SYSTEM SystemTests
  (* Version 1.0, 2018-08-29, Alois Zoitl, Johannes Kepler University, initial API and implementation and/or initial documentation *)
  APPLICATION Timing (* Small test application for measuring the execution time of a few fbs for evaluating runtime performance *)
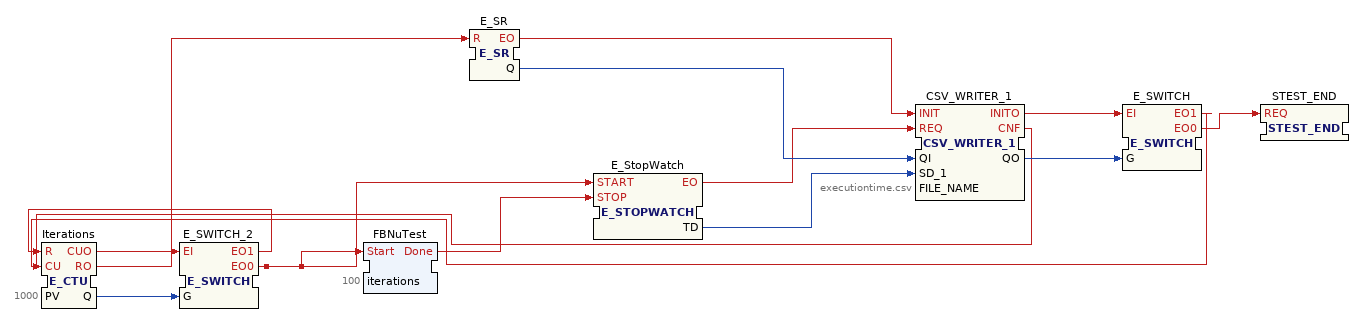
    FBS
      CSV_WRITER_1 : CSV_WRITER_1(FILE_NAME := executiontime.csv);
      E_SR : E_SR;
      E_SWITCH_2 : E_SWITCH;
      Iterations : E_CTU(PV := 1000);
      STEST_END : STEST_END;
      E_SWITCH : E_SWITCH;
      E_StopWatch : E_STOPWATCH;
    END_FBS
    SUBAPPLICATION FBNuTest(iterations := 100)
      EVENT_INPUT
        Start;
      END_EVENT
      EVENT_OUTPUT
        Done;
      END_EVENT
      VAR_INPUT
        iterations : UINT := 100;
      END_VAR
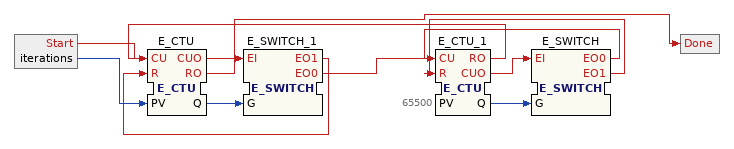
      FBS
        E_CTU : E_CTU;
        E_SWITCH_1 : E_SWITCH;
        E_SWITCH : E_SWITCH;
        E_CTU_1 : E_CTU(PV := 65500);
      END_FBS
      EVENT_CONNECTIONS
        E_CTU_1.RO TO E_CTU.CU;
        E_SWITCH_1.EO1 TO E_CTU.R;
        E_CTU.CUO TO E_SWITCH_1.EI;
        E_SWITCH_1.EO0 TO E_CTU_1.CU;
        E_CTU_1.CUO TO E_SWITCH.EI;
        E_SWITCH.EO0 TO E_CTU_1.CU;
        E_SWITCH.EO1 TO E_CTU_1.R;
        Start TO E_CTU.CU;
        E_CTU.RO TO Done;
      END_CONNECTIONS
      DATA_CONNECTIONS
        E_CTU.Q TO E_SWITCH_1.G;
        E_CTU_1.Q TO E_SWITCH.G;
        iterations TO E_CTU.PV;
      END_CONNECTIONS
    END_SUBAPPLICATION
    EVENT_CONNECTIONS
      E_SR.EO TO CSV_WRITER_1.INIT;
      Iterations.CUO TO E_SWITCH_2.EI;
      E_SWITCH_2.EO1 TO Iterations.R;
      Iterations.RO TO E_SR.R;
      E_SWITCH_2.EO0 TO FBNuTest.Start;
      E_SWITCH.EO1 TO Iterations.CU;
      E_SWITCH.EO0 TO STEST_END.REQ;
      CSV_WRITER_1.INITO TO E_SWITCH.EI;
      E_SWITCH_2.EO0 TO E_StopWatch.START;
      FBNuTest.Done TO E_StopWatch.STOP;
      E_StopWatch.EO TO CSV_WRITER_1.REQ;
      CSV_WRITER_1.CNF TO Iterations.CU;
    END_CONNECTIONS
    DATA_CONNECTIONS
      E_SR.Q TO CSV_WRITER_1.QI;
      Iterations.Q TO E_SWITCH_2.G;
      CSV_WRITER_1.QO TO E_SWITCH.G;
      E_StopWatch.TD TO CSV_WRITER_1.SD_1;
    END_CONNECTIONS
  END_APPLICATION
  APPLICATION Soft_Pass_Example
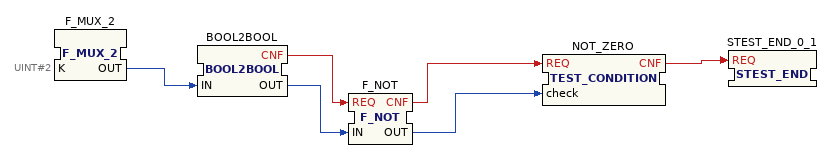
    FBS
      NOT_ZERO : TEST_CONDITION;
      STEST_END_0_1 : STEST_END;
      F_MUX_2 : F_MUX_2(K := UINT#2);
      F_NOT : F_NOT;
      BOOL2BOOL : BOOL2BOOL;
    END_FBS
    EVENT_CONNECTIONS
      F_NOT.CNF TO NOT_ZERO.REQ;
      NOT_ZERO.CNF TO STEST_END_0_1.REQ;
      BOOL2BOOL.CNF TO F_NOT.REQ;
    END_CONNECTIONS
    DATA_CONNECTIONS
      F_MUX_2.OUT TO BOOL2BOOL.IN;
      F_NOT.OUT TO NOT_ZERO.check;
      BOOL2BOOL.OUT TO F_NOT.IN;
    END_CONNECTIONS
  END_APPLICATION
  APPLICATION Fail_Example
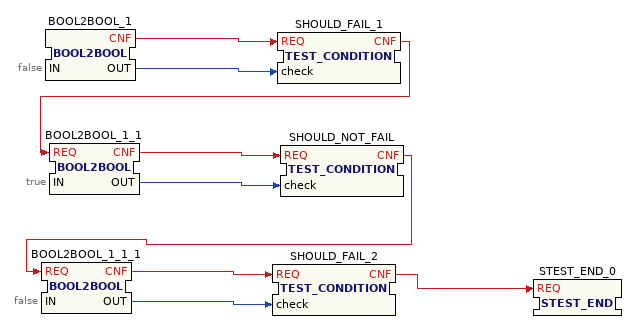
    FBS
      STEST_END_0 : STEST_END;
      BOOL2BOOL_1_1_1 : BOOL2BOOL(IN := false);
      SHOULD_FAIL_1 : TEST_CONDITION;
      BOOL2BOOL_1 : BOOL2BOOL(IN := false);
      SHOULD_NOT_FAIL : TEST_CONDITION;
      BOOL2BOOL_1_1 : BOOL2BOOL(IN := true);
      SHOULD_FAIL_2 : TEST_CONDITION;
    END_FBS
    EVENT_CONNECTIONS
      BOOL2BOOL_1.CNF TO SHOULD_FAIL_1.REQ;
      SHOULD_FAIL_2.CNF TO STEST_END_0.REQ;
      SHOULD_FAIL_1.CNF TO BOOL2BOOL_1_1.REQ;
      SHOULD_NOT_FAIL.CNF TO BOOL2BOOL_1_1_1.REQ;
      BOOL2BOOL_1_1_1.CNF TO SHOULD_FAIL_2.REQ;
      BOOL2BOOL_1_1.CNF TO SHOULD_NOT_FAIL.REQ;
    END_CONNECTIONS
    DATA_CONNECTIONS
      BOOL2BOOL_1_1.OUT TO SHOULD_NOT_FAIL.check;
      BOOL2BOOL_1.OUT TO SHOULD_FAIL_1.check;
      BOOL2BOOL_1_1_1.OUT TO SHOULD_FAIL_2.check;
    END_CONNECTIONS
  END_APPLICATION
  APPLICATION Hard_Pass_Example
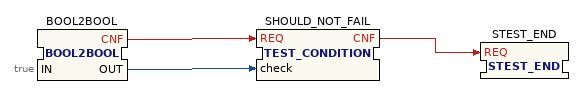
    FBS
      STEST_END : STEST_END;
      BOOL2BOOL : BOOL2BOOL(IN := true);
      SHOULD_NOT_FAIL : TEST_CONDITION;
    END_FBS
    EVENT_CONNECTIONS
      BOOL2BOOL.CNF TO SHOULD_NOT_FAIL.REQ;
      SHOULD_NOT_FAIL.CNF TO STEST_END.REQ;
    END_CONNECTIONS
    DATA_CONNECTIONS
      BOOL2BOOL.OUT TO SHOULD_NOT_FAIL.check;
    END_CONNECTIONS
  END_APPLICATION
  APPLICATION DeInitCommFB
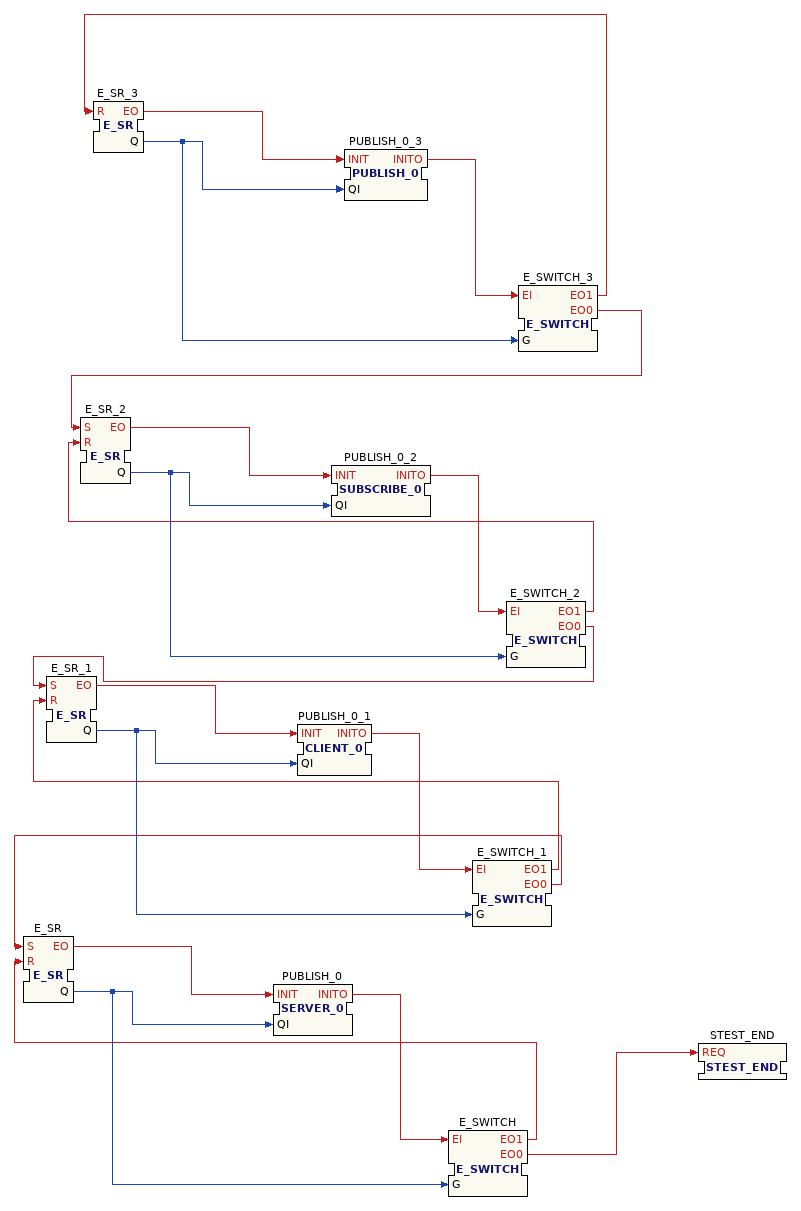
    FBS
      E_SR : E_SR;
      E_SWITCH : E_SWITCH;
      STEST_END : STEST_END;
      PUBLISH_0 : SERVER_0;
      E_SWITCH_1 : E_SWITCH;
      E_SR_1 : E_SR;
      E_SWITCH_2 : E_SWITCH;
      E_SR_2 : E_SR;
      E_SR_3 : E_SR;
      E_SWITCH_3 : E_SWITCH;
      PUBLISH_0_3 : PUBLISH_0;
      PUBLISH_0_2 : SUBSCRIBE_0;
      PUBLISH_0_1 : CLIENT_0;
    END_FBS
    EVENT_CONNECTIONS
      PUBLISH_0.INITO TO E_SWITCH.EI;
      E_SR_3.EO TO PUBLISH_0_3.INIT;
      PUBLISH_0_3.INITO TO E_SWITCH_3.EI;
      E_SR_2.EO TO PUBLISH_0_2.INIT;
      PUBLISH_0_2.INITO TO E_SWITCH_2.EI;
      E_SR_1.EO TO PUBLISH_0_1.INIT;
      PUBLISH_0_1.INITO TO E_SWITCH_1.EI;
      E_SWITCH_3.EO1 TO E_SR_3.R;
      E_SWITCH_3.EO0 TO E_SR_2.S;
      E_SWITCH_2.EO1 TO E_SR_2.R;
      E_SWITCH_2.EO0 TO E_SR_1.S;
      E_SWITCH_1.EO1 TO E_SR_1.R;
      E_SWITCH_1.EO0 TO E_SR.S;
      E_SWITCH.EO1 TO E_SR.R;
      E_SWITCH.EO0 TO STEST_END.REQ;
      E_SR.EO TO PUBLISH_0.INIT;
    END_CONNECTIONS
    DATA_CONNECTIONS
      E_SR.Q TO E_SWITCH.G;
      E_SR.Q TO PUBLISH_0.QI;
      E_SR_1.Q TO E_SWITCH_1.G;
      E_SR_2.Q TO E_SWITCH_2.G;
      E_SR_3.Q TO E_SWITCH_3.G;
      E_SR_3.Q TO PUBLISH_0_3.QI;
      E_SR_2.Q TO PUBLISH_0_2.QI;
      E_SR_1.Q TO PUBLISH_0_1.QI;
    END_CONNECTIONS
  END_APPLICATION
  APPLICATION simpleCommunicationTest
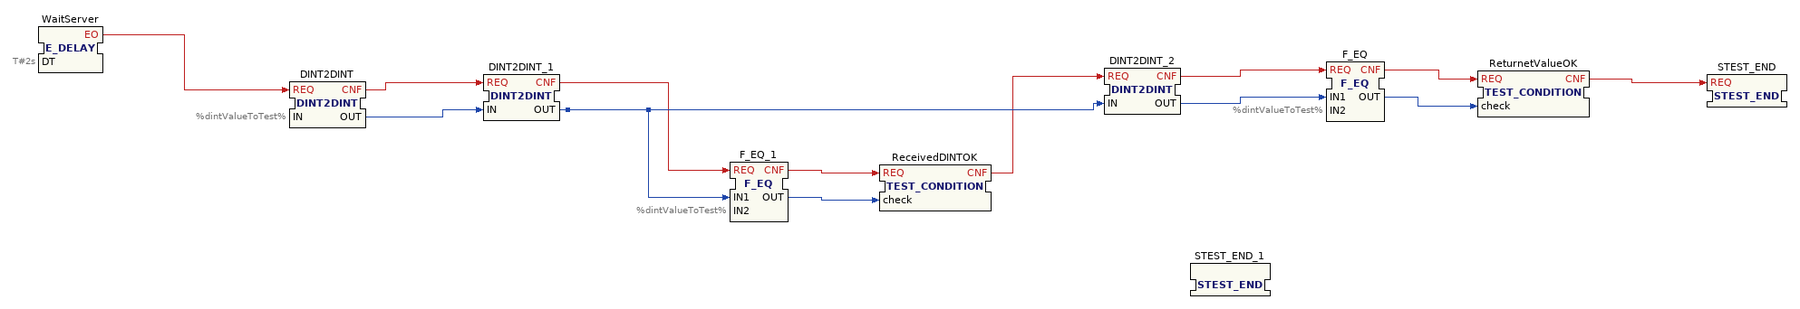
    FBS
      WaitServer : E_DELAY(DT := T#2s);
      ReturnetValueOK : TEST_CONDITION;
      F_EQ_1 : F_EQ(IN2 := %dintValueToTest%);
      F_EQ : F_EQ(IN2 := %dintValueToTest%);
      DINT2DINT_2 : DINT2DINT;
      DINT2DINT_1 : DINT2DINT;
      STEST_END : STEST_END;
      DINT2DINT : DINT2DINT(IN := %dintValueToTest%);
      ReceivedDINTOK : TEST_CONDITION;
      STEST_END_1 : STEST_END;
    END_FBS
    EVENT_CONNECTIONS
      DINT2DINT_1.CNF TO F_EQ_1.REQ;
      DINT2DINT.CNF TO DINT2DINT_1.REQ;
      ReceivedDINTOK.CNF TO DINT2DINT_2.REQ;
      F_EQ_1.CNF TO ReceivedDINTOK.REQ;
      F_EQ.CNF TO ReturnetValueOK.REQ;
      ReturnetValueOK.CNF TO STEST_END.REQ;
      DINT2DINT_2.CNF TO F_EQ.REQ;
      WaitServer.EO TO DINT2DINT.REQ;
    END_CONNECTIONS
    DATA_CONNECTIONS
      F_EQ_1.OUT TO ReceivedDINTOK.check;
      DINT2DINT_1.OUT TO DINT2DINT_2.IN;
      DINT2DINT.OUT TO DINT2DINT_1.IN;
      F_EQ.OUT TO ReturnetValueOK.check;
      DINT2DINT_1.OUT TO F_EQ_1.IN1;
      DINT2DINT_2.OUT TO F_EQ.IN1;
    END_CONNECTIONS
  END_APPLICATION
  APPLICATION CSVWriterTests
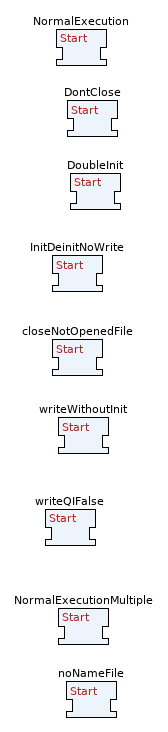
    SUBAPPLICATION NormalExecution
      EVENT_INPUT
        Start;
      END_EVENT
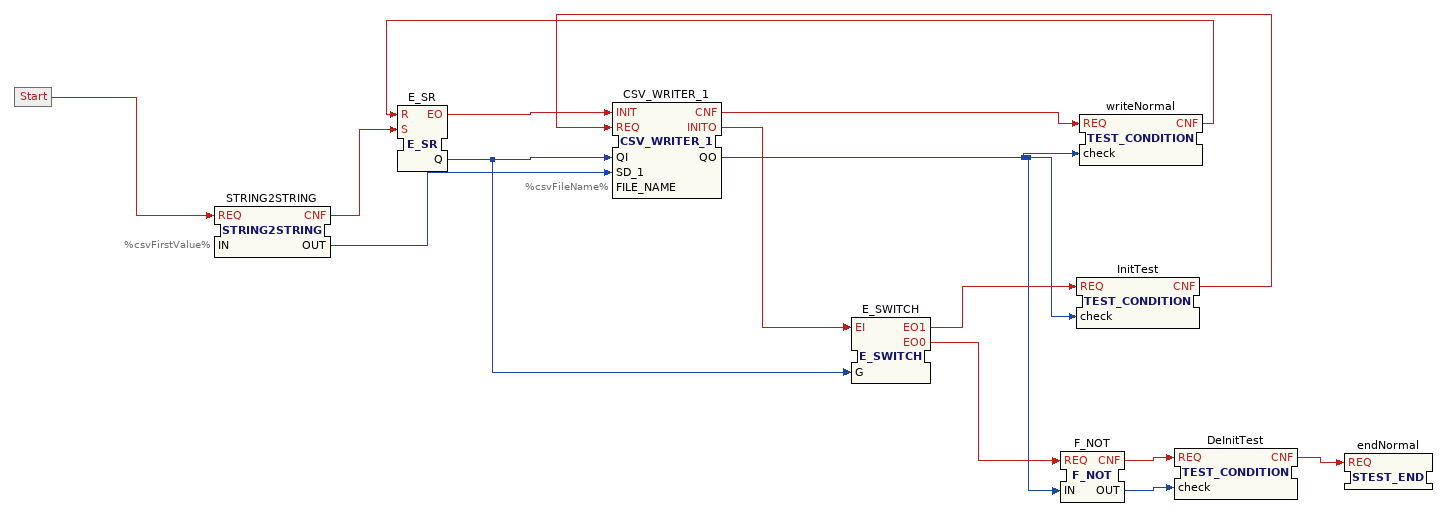
      FBS
        writeNormal : TEST_CONDITION;
        CSV_WRITER_1 : CSV_WRITER_1(FILE_NAME := %csvFileName%);
        InitTest : TEST_CONDITION;
        STRING2STRING : STRING2STRING(IN := %csvFirstValue%);
        DeInitTest : TEST_CONDITION;
        endNormal : STEST_END;
        F_NOT : F_NOT;
        E_SWITCH : E_SWITCH;
        E_SR : E_SR;
      END_FBS
      EVENT_CONNECTIONS
        CSV_WRITER_1.CNF TO writeNormal.REQ;
        writeNormal.CNF TO E_SR.R;
        E_SR.EO TO CSV_WRITER_1.INIT;
        InitTest.CNF TO CSV_WRITER_1.REQ;
        CSV_WRITER_1.INITO TO E_SWITCH.EI;
        E_SWITCH.EO1 TO InitTest.REQ;
        STRING2STRING.CNF TO E_SR.S;
        F_NOT.CNF TO DeInitTest.REQ;
        DeInitTest.CNF TO endNormal.REQ;
        E_SWITCH.EO0 TO F_NOT.REQ;
        Start TO STRING2STRING.REQ;
      END_CONNECTIONS
      DATA_CONNECTIONS
        CSV_WRITER_1.QO TO writeNormal.check;
        E_SR.Q TO CSV_WRITER_1.QI;
        STRING2STRING.OUT TO CSV_WRITER_1.SD_1;
        CSV_WRITER_1.QO TO InitTest.check;
        CSV_WRITER_1.QO TO F_NOT.IN;
        F_NOT.OUT TO DeInitTest.check;
        E_SR.Q TO E_SWITCH.G;
      END_CONNECTIONS
    END_SUBAPPLICATION
    SUBAPPLICATION DontClose
      EVENT_INPUT
        Start;
      END_EVENT
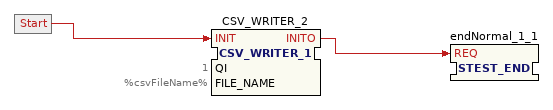
      FBS
        CSV_WRITER_2 : CSV_WRITER_1(QI := 1, FILE_NAME := %csvFileName%);
        endNormal_1_1 : STEST_END;
      END_FBS
      EVENT_CONNECTIONS
        CSV_WRITER_2.INITO TO endNormal_1_1.REQ;
        Start TO CSV_WRITER_2.INIT;
      END_CONNECTIONS
    END_SUBAPPLICATION
    SUBAPPLICATION DoubleInit
      EVENT_INPUT
        Start;
      END_EVENT
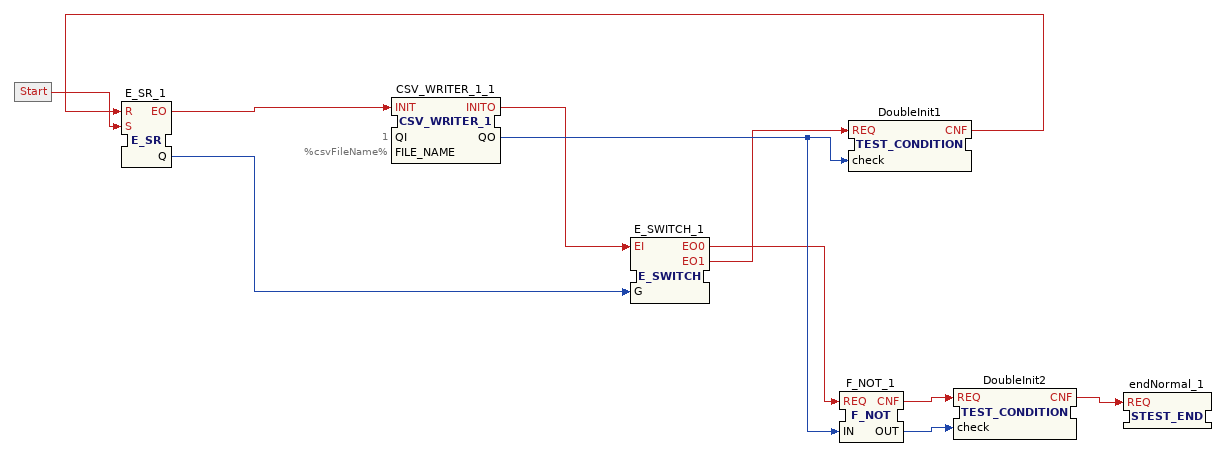
      FBS
        F_NOT_1 : F_NOT;
        E_SR_1 : E_SR;
        DoubleInit1 : TEST_CONDITION;
        CSV_WRITER_1_1 : CSV_WRITER_1(QI := 1, FILE_NAME := %csvFileName%);
        E_SWITCH_1 : E_SWITCH;
        endNormal_1 : STEST_END;
        DoubleInit2 : TEST_CONDITION;
      END_FBS
      EVENT_CONNECTIONS
        E_SWITCH_1.EO0 TO F_NOT_1.REQ;
        F_NOT_1.CNF TO DoubleInit2.REQ;
        DoubleInit1.CNF TO E_SR_1.R;
        E_SR_1.EO TO CSV_WRITER_1_1.INIT;
        E_SWITCH_1.EO1 TO DoubleInit1.REQ;
        CSV_WRITER_1_1.INITO TO E_SWITCH_1.EI;
        DoubleInit2.CNF TO endNormal_1.REQ;
        Start TO E_SR_1.S;
      END_CONNECTIONS
      DATA_CONNECTIONS
        CSV_WRITER_1_1.QO TO F_NOT_1.IN;
        F_NOT_1.OUT TO DoubleInit2.check;
        E_SR_1.Q TO E_SWITCH_1.G;
        CSV_WRITER_1_1.QO TO DoubleInit1.check;
      END_CONNECTIONS
    END_SUBAPPLICATION
    SUBAPPLICATION InitDeinitNoWrite
      EVENT_INPUT
        Start;
      END_EVENT
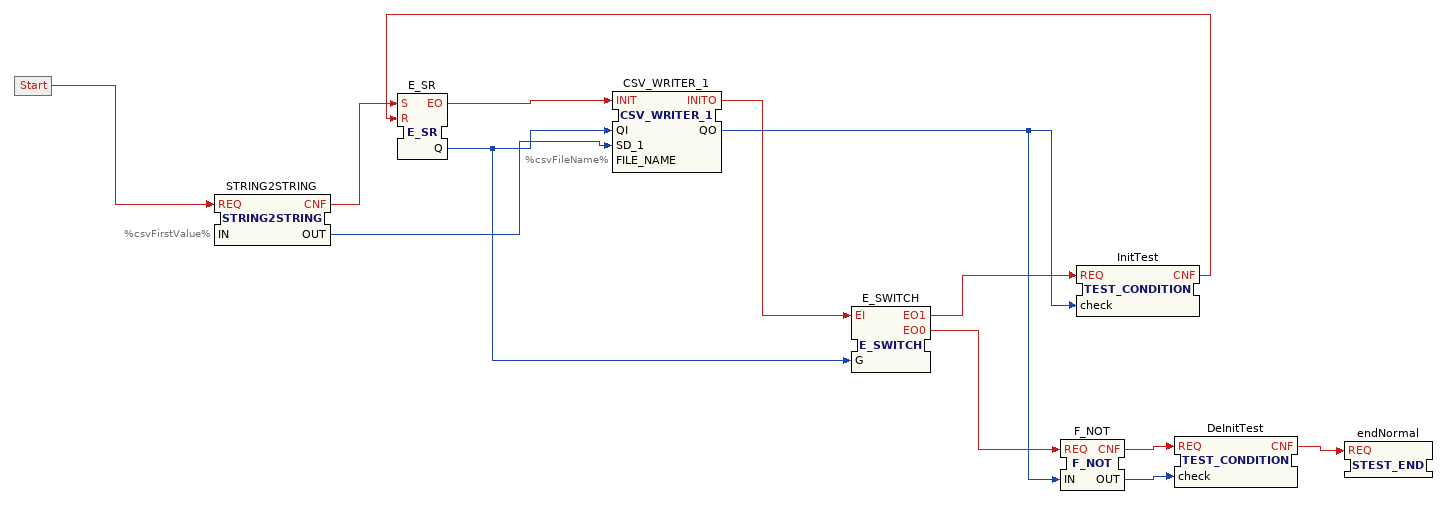
      FBS
        CSV_WRITER_1 : CSV_WRITER_1(FILE_NAME := %csvFileName%);
        InitTest : TEST_CONDITION;
        STRING2STRING : STRING2STRING(IN := %csvFirstValue%);
        DeInitTest : TEST_CONDITION;
        endNormal : STEST_END;
        F_NOT : F_NOT;
        E_SWITCH : E_SWITCH;
        E_SR : E_SR;
      END_FBS
      EVENT_CONNECTIONS
        E_SR.EO TO CSV_WRITER_1.INIT;
        CSV_WRITER_1.INITO TO E_SWITCH.EI;
        E_SWITCH.EO1 TO InitTest.REQ;
        STRING2STRING.CNF TO E_SR.S;
        F_NOT.CNF TO DeInitTest.REQ;
        DeInitTest.CNF TO endNormal.REQ;
        E_SWITCH.EO0 TO F_NOT.REQ;
        Start TO STRING2STRING.REQ;
        InitTest.CNF TO E_SR.R;
      END_CONNECTIONS
      DATA_CONNECTIONS
        E_SR.Q TO CSV_WRITER_1.QI;
        STRING2STRING.OUT TO CSV_WRITER_1.SD_1;
        CSV_WRITER_1.QO TO InitTest.check;
        CSV_WRITER_1.QO TO F_NOT.IN;
        F_NOT.OUT TO DeInitTest.check;
        E_SR.Q TO E_SWITCH.G;
      END_CONNECTIONS
    END_SUBAPPLICATION
    SUBAPPLICATION closeNotOpenedFile
      EVENT_INPUT
        Start;
      END_EVENT
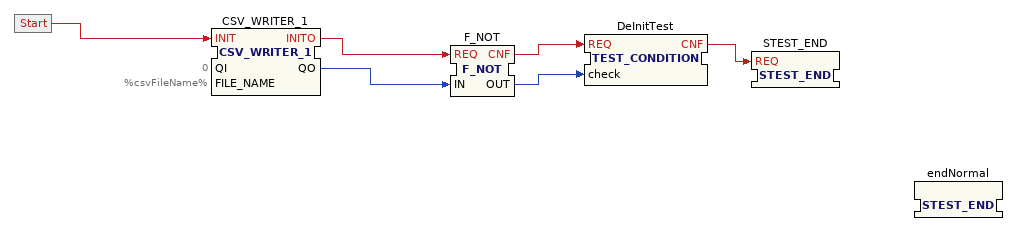
      FBS
        CSV_WRITER_1 : CSV_WRITER_1(QI := 0, FILE_NAME := %csvFileName%);
        DeInitTest : TEST_CONDITION;
        endNormal : STEST_END;
        F_NOT : F_NOT;
        STEST_END : STEST_END;
      END_FBS
      EVENT_CONNECTIONS
        F_NOT.CNF TO DeInitTest.REQ;
        CSV_WRITER_1.INITO TO F_NOT.REQ;
        Start TO CSV_WRITER_1.INIT;
        DeInitTest.CNF TO STEST_END.REQ;
      END_CONNECTIONS
      DATA_CONNECTIONS
        F_NOT.OUT TO DeInitTest.check;
        CSV_WRITER_1.QO TO F_NOT.IN;
      END_CONNECTIONS
    END_SUBAPPLICATION
    SUBAPPLICATION writeWithoutInit
      EVENT_INPUT
        Start;
      END_EVENT
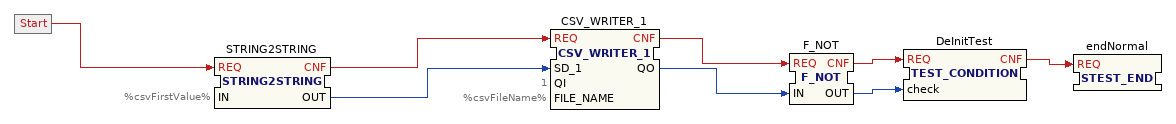
      FBS
        CSV_WRITER_1 : CSV_WRITER_1(QI := 1, FILE_NAME := %csvFileName%);
        STRING2STRING : STRING2STRING(IN := %csvFirstValue%);
        DeInitTest : TEST_CONDITION;
        endNormal : STEST_END;
        F_NOT : F_NOT;
      END_FBS
      EVENT_CONNECTIONS
        F_NOT.CNF TO DeInitTest.REQ;
        DeInitTest.CNF TO endNormal.REQ;
        Start TO STRING2STRING.REQ;
        STRING2STRING.CNF TO CSV_WRITER_1.REQ;
        CSV_WRITER_1.CNF TO F_NOT.REQ;
      END_CONNECTIONS
      DATA_CONNECTIONS
        STRING2STRING.OUT TO CSV_WRITER_1.SD_1;
        CSV_WRITER_1.QO TO F_NOT.IN;
        F_NOT.OUT TO DeInitTest.check;
      END_CONNECTIONS
    END_SUBAPPLICATION
    SUBAPPLICATION writeQIFalse
      EVENT_INPUT
        Start;
      END_EVENT
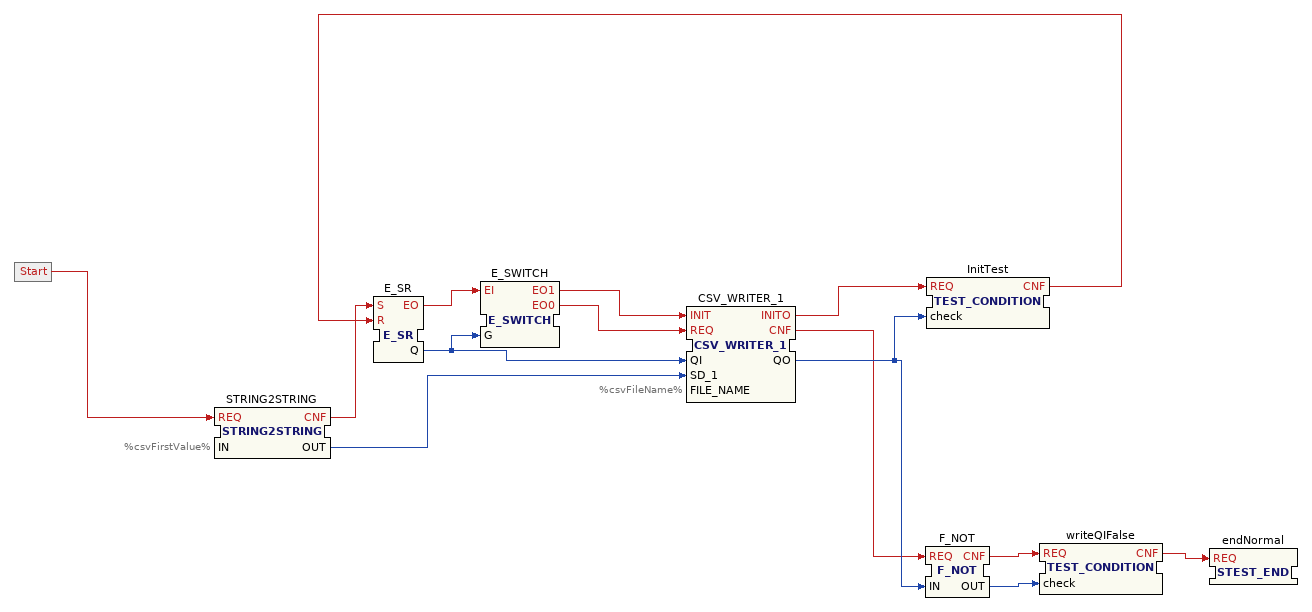
      FBS
        CSV_WRITER_1 : CSV_WRITER_1(FILE_NAME := %csvFileName%);
        InitTest : TEST_CONDITION;
        STRING2STRING : STRING2STRING(IN := %csvFirstValue%);
        writeQIFalse : TEST_CONDITION;
        endNormal : STEST_END;
        F_NOT : F_NOT;
        E_SR : E_SR;
        E_SWITCH : E_SWITCH;
      END_FBS
      EVENT_CONNECTIONS
        STRING2STRING.CNF TO E_SR.S;
        F_NOT.CNF TO writeQIFalse.REQ;
        writeQIFalse.CNF TO endNormal.REQ;
        Start TO STRING2STRING.REQ;
        CSV_WRITER_1.INITO TO InitTest.REQ;
        InitTest.CNF TO E_SR.R;
        E_SWITCH.EO1 TO CSV_WRITER_1.INIT;
        E_SWITCH.EO0 TO CSV_WRITER_1.REQ;
        E_SR.EO TO E_SWITCH.EI;
        CSV_WRITER_1.CNF TO F_NOT.REQ;
      END_CONNECTIONS
      DATA_CONNECTIONS
        E_SR.Q TO CSV_WRITER_1.QI;
        STRING2STRING.OUT TO CSV_WRITER_1.SD_1;
        CSV_WRITER_1.QO TO InitTest.check;
        CSV_WRITER_1.QO TO F_NOT.IN;
        F_NOT.OUT TO writeQIFalse.check;
        E_SR.Q TO E_SWITCH.G;
      END_CONNECTIONS
    END_SUBAPPLICATION
    SUBAPPLICATION NormalExecutionMultiple
      EVENT_INPUT
        Start;
      END_EVENT
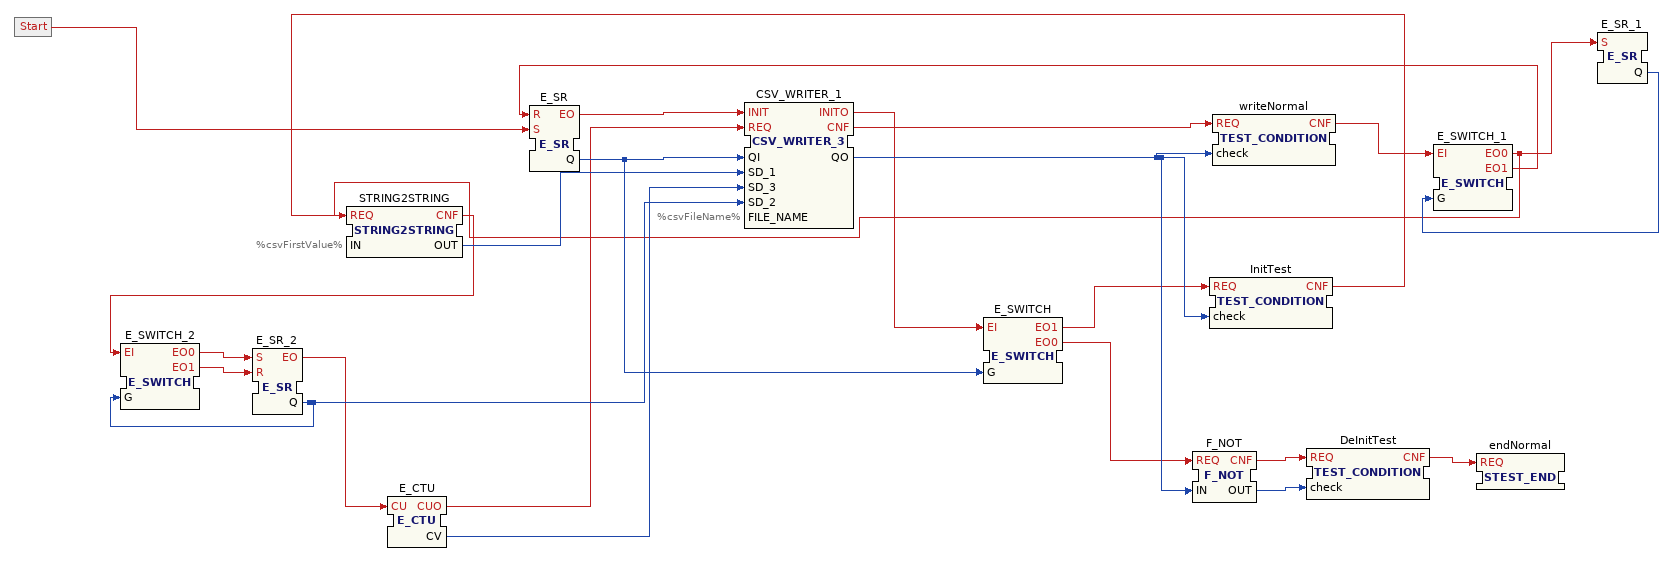
      FBS
        writeNormal : TEST_CONDITION;
        InitTest : TEST_CONDITION;
        STRING2STRING : STRING2STRING(IN := %csvFirstValue%);
        DeInitTest : TEST_CONDITION;
        endNormal : STEST_END;
        F_NOT : F_NOT;
        E_SWITCH : E_SWITCH;
        E_SR : E_SR;
        CSV_WRITER_1 : CSV_WRITER_3(FILE_NAME := %csvFileName%);
        E_SR_1 : E_SR;
        E_SWITCH_1 : E_SWITCH;
        E_SR_2 : E_SR;
        E_SWITCH_2 : E_SWITCH;
        E_CTU : E_CTU;
      END_FBS
      EVENT_CONNECTIONS
        E_SWITCH.EO1 TO InitTest.REQ;
        F_NOT.CNF TO DeInitTest.REQ;
        DeInitTest.CNF TO endNormal.REQ;
        E_SWITCH.EO0 TO F_NOT.REQ;
        E_SR.EO TO CSV_WRITER_1.INIT;
        CSV_WRITER_1.INITO TO E_SWITCH.EI;
        CSV_WRITER_1.CNF TO writeNormal.REQ;
        writeNormal.CNF TO E_SWITCH_1.EI;
        E_SWITCH_1.EO0 TO E_SR_1.S;
        E_SWITCH_1.EO1 TO E_SR.R;
        Start TO E_SR.S;
        InitTest.CNF TO STRING2STRING.REQ;
        E_SWITCH_1.EO0 TO STRING2STRING.REQ;
        STRING2STRING.CNF TO E_SWITCH_2.EI;
        E_SWITCH_2.EO0 TO E_SR_2.S;
        E_SWITCH_2.EO1 TO E_SR_2.R;
        E_CTU.CUO TO CSV_WRITER_1.REQ;
        E_SR_2.EO TO E_CTU.CU;
      END_CONNECTIONS
      DATA_CONNECTIONS
        F_NOT.OUT TO DeInitTest.check;
        E_SR.Q TO E_SWITCH.G;
        E_SR.Q TO CSV_WRITER_1.QI;
        STRING2STRING.OUT TO CSV_WRITER_1.SD_1;
        CSV_WRITER_1.QO TO InitTest.check;
        CSV_WRITER_1.QO TO F_NOT.IN;
        CSV_WRITER_1.QO TO writeNormal.check;
        E_SR_1.Q TO E_SWITCH_1.G;
        E_SR_2.Q TO E_SWITCH_2.G;
        E_CTU.CV TO CSV_WRITER_1.SD_3;
        E_SR_2.Q TO CSV_WRITER_1.SD_2;
      END_CONNECTIONS
    END_SUBAPPLICATION
    SUBAPPLICATION noNameFile
      EVENT_INPUT
        Start;
      END_EVENT
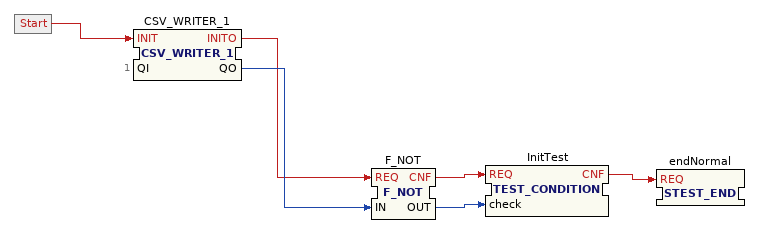
      FBS
        CSV_WRITER_1 : CSV_WRITER_1(QI := 1);
        InitTest : TEST_CONDITION;
        endNormal : STEST_END;
        F_NOT : F_NOT;
      END_FBS
      EVENT_CONNECTIONS
        F_NOT.CNF TO InitTest.REQ;
        InitTest.CNF TO endNormal.REQ;
        Start TO CSV_WRITER_1.INIT;
        CSV_WRITER_1.INITO TO F_NOT.REQ;
      END_CONNECTIONS
      DATA_CONNECTIONS
        CSV_WRITER_1.QO TO F_NOT.IN;
        F_NOT.OUT TO InitTest.check;
      END_CONNECTIONS
    END_SUBAPPLICATION
  END_APPLICATION
  APPLICATION MultiDevice
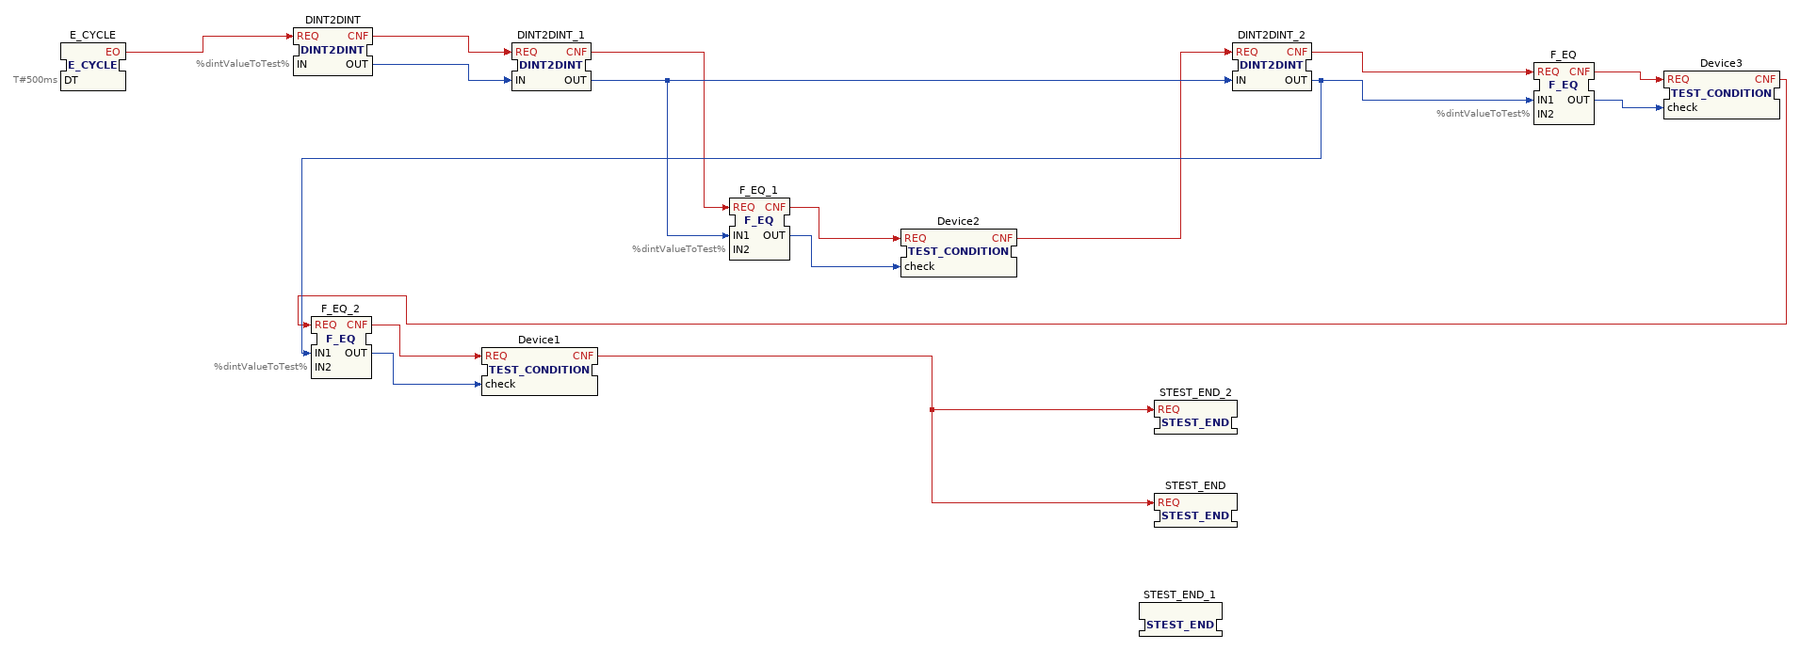
    FBS
      F_EQ_1 : F_EQ(IN2 := %dintValueToTest%);
      STEST_END : STEST_END;
      DINT2DINT_1 : DINT2DINT;
      DINT2DINT_2 : DINT2DINT;
      DINT2DINT : DINT2DINT(IN := %dintValueToTest%);
      Device3 : TEST_CONDITION;
      F_EQ : F_EQ(IN2 := %dintValueToTest%);
      Device2 : TEST_CONDITION;
      STEST_END_1 : STEST_END;
      E_CYCLE : E_CYCLE(DT := T#500ms);
      STEST_END_2 : STEST_END;
      F_EQ_2 : F_EQ(IN2 := %dintValueToTest%);
      Device1 : TEST_CONDITION;
    END_FBS
    EVENT_CONNECTIONS
      DINT2DINT.CNF TO DINT2DINT_1.REQ;
      F_EQ_1.CNF TO Device2.REQ;
      F_EQ.CNF TO Device3.REQ;
      DINT2DINT_2.CNF TO F_EQ.REQ;
      E_CYCLE.EO TO DINT2DINT.REQ;
      DINT2DINT_1.CNF TO F_EQ_1.REQ;
      Device2.CNF TO DINT2DINT_2.REQ;
      F_EQ_2.CNF TO Device1.REQ;
      Device3.CNF TO F_EQ_2.REQ;
      Device1.CNF TO STEST_END.REQ;
      Device1.CNF TO STEST_END_2.REQ;
    END_CONNECTIONS
    DATA_CONNECTIONS
      DINT2DINT_2.OUT TO F_EQ.IN1;
      DINT2DINT_1.OUT TO F_EQ_1.IN1;
      DINT2DINT_1.OUT TO DINT2DINT_2.IN;
      F_EQ_1.OUT TO Device2.check;
      F_EQ.OUT TO Device3.check;
      DINT2DINT.OUT TO DINT2DINT_1.IN;
      F_EQ_2.OUT TO Device1.check;
      DINT2DINT_2.OUT TO F_EQ_2.IN1;
    END_CONNECTIONS
  END_APPLICATION
  DEVICE DuT : FORTE_PC(MGR_ID := "localhost:61499")
    {SET_ATTRIBUTE(Profile, HOLOBLOC)} (* device profile *)
    RESOURCE TimingTestRes : EMB_RES
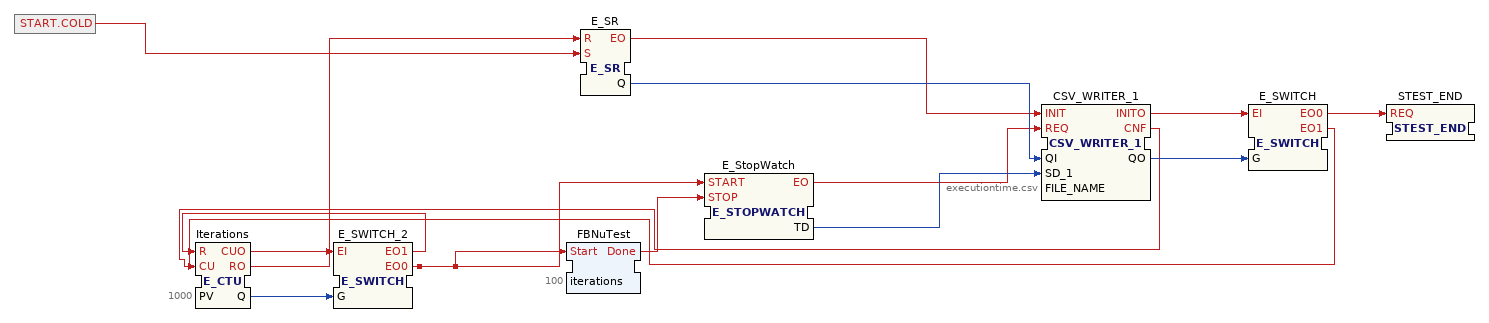
      FBS
        CSV_WRITER_1 : CSV_WRITER_1(FILE_NAME := executiontime.csv);
        E_SR : E_SR;
        E_SWITCH_2 : E_SWITCH;
        Iterations : E_CTU(PV := 1000);
        STEST_END : STEST_END;
        E_SWITCH : E_SWITCH;
        E_StopWatch : E_STOPWATCH;
      END_FBS
      SUBAPPLICATION FBNuTest(iterations := 100)
        EVENT_INPUT
          Start;
        END_EVENT
        EVENT_OUTPUT
          Done;
        END_EVENT
        VAR_INPUT
          iterations : ANY_MAGNITUDE := 100;
        END_VAR
      END_SUBAPPLICATION
      EVENT_CONNECTIONS
        E_SR.EO TO CSV_WRITER_1.INIT;
        E_SWITCH_2.EO1 TO Iterations.R;
        Iterations.CUO TO E_SWITCH_2.EI;
        Iterations.RO TO E_SR.R;
        E_SWITCH_2.EO0 TO FBNuTest.Start;
        START.COLD TO E_SR.S;
        CSV_WRITER_1.INITO TO E_SWITCH.EI;
        E_SWITCH.EO0 TO STEST_END.REQ;
        E_SWITCH.EO1 TO Iterations.CU;
        E_SWITCH_2.EO0 TO E_StopWatch.START;
        FBNuTest.Done TO E_StopWatch.STOP;
        E_StopWatch.EO TO CSV_WRITER_1.REQ;
        CSV_WRITER_1.CNF TO Iterations.CU;
      END_CONNECTIONS
      DATA_CONNECTIONS
        E_SR.Q TO CSV_WRITER_1.QI;
        Iterations.Q TO E_SWITCH_2.G;
        CSV_WRITER_1.QO TO E_SWITCH.G;
        E_StopWatch.TD TO CSV_WRITER_1.SD_1;
      END_CONNECTIONS
    END_RESOURCE
    RESOURCE Hard_Pass_Example : EMB_RES
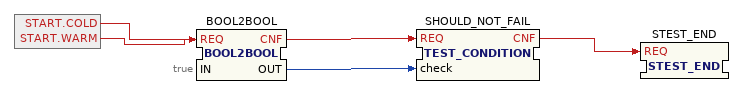
      FBS
        STEST_END : STEST_END;
        SHOULD_NOT_FAIL : TEST_CONDITION;
        BOOL2BOOL : BOOL2BOOL(IN := true);
      END_FBS
      EVENT_CONNECTIONS
        SHOULD_NOT_FAIL.CNF TO STEST_END.REQ;
        BOOL2BOOL.CNF TO SHOULD_NOT_FAIL.REQ;
        START.COLD TO BOOL2BOOL.REQ;
        START.WARM TO BOOL2BOOL.REQ;
      END_CONNECTIONS
      DATA_CONNECTIONS
        BOOL2BOOL.OUT TO SHOULD_NOT_FAIL.check;
      END_CONNECTIONS
    END_RESOURCE
    RESOURCE Soft_Pass_Example : EMB_RES
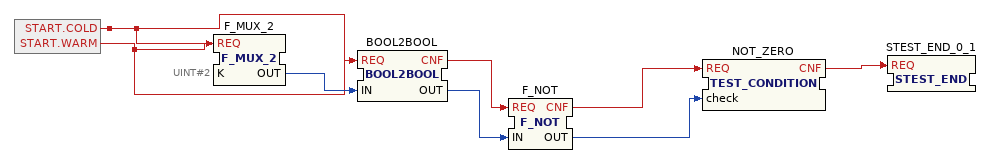
      FBS
        NOT_ZERO : TEST_CONDITION;
        F_NOT : F_NOT;
        BOOL2BOOL : BOOL2BOOL;
        STEST_END_0_1 : STEST_END;
        F_MUX_2 : F_MUX_2(K := UINT#2);
      END_FBS
      EVENT_CONNECTIONS
        F_NOT.CNF TO NOT_ZERO.REQ;
        BOOL2BOOL.CNF TO F_NOT.REQ;
        NOT_ZERO.CNF TO STEST_END_0_1.REQ;
        START.COLD TO F_MUX_2.REQ;
        START.WARM TO F_MUX_2.REQ;
        START.COLD TO BOOL2BOOL.REQ;
        START.WARM TO BOOL2BOOL.REQ;
      END_CONNECTIONS
      DATA_CONNECTIONS
        F_NOT.OUT TO NOT_ZERO.check;
        BOOL2BOOL.OUT TO F_NOT.IN;
        F_MUX_2.OUT TO BOOL2BOOL.IN;
      END_CONNECTIONS
    END_RESOURCE
    RESOURCE Fail_Example : EMB_RES
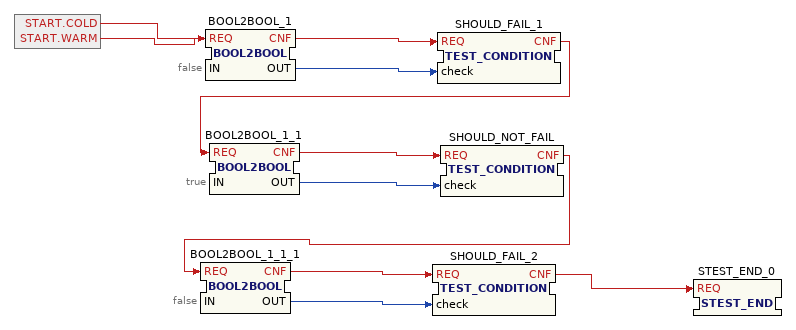
      FBS
        BOOL2BOOL_1_1_1 : BOOL2BOOL(IN := false);
        BOOL2BOOL_1 : BOOL2BOOL(IN := false);
        BOOL2BOOL_1_1 : BOOL2BOOL(IN := true);
        STEST_END_0 : STEST_END;
        SHOULD_FAIL_1 : TEST_CONDITION;
        SHOULD_FAIL_2 : TEST_CONDITION;
        SHOULD_NOT_FAIL : TEST_CONDITION;
      END_FBS
      EVENT_CONNECTIONS
        BOOL2BOOL_1.CNF TO SHOULD_FAIL_1.REQ;
        SHOULD_FAIL_1.CNF TO BOOL2BOOL_1_1.REQ;
        BOOL2BOOL_1_1_1.CNF TO SHOULD_FAIL_2.REQ;
        SHOULD_FAIL_2.CNF TO STEST_END_0.REQ;
        BOOL2BOOL_1_1.CNF TO SHOULD_NOT_FAIL.REQ;
        SHOULD_NOT_FAIL.CNF TO BOOL2BOOL_1_1_1.REQ;
        START.COLD TO BOOL2BOOL_1.REQ;
        START.WARM TO BOOL2BOOL_1.REQ;
      END_CONNECTIONS
      DATA_CONNECTIONS
        BOOL2BOOL_1.OUT TO SHOULD_FAIL_1.check;
        BOOL2BOOL_1_1_1.OUT TO SHOULD_FAIL_2.check;
        BOOL2BOOL_1_1.OUT TO SHOULD_NOT_FAIL.check;
      END_CONNECTIONS
    END_RESOURCE
    RESOURCE DeInitCommFB : EMB_RES
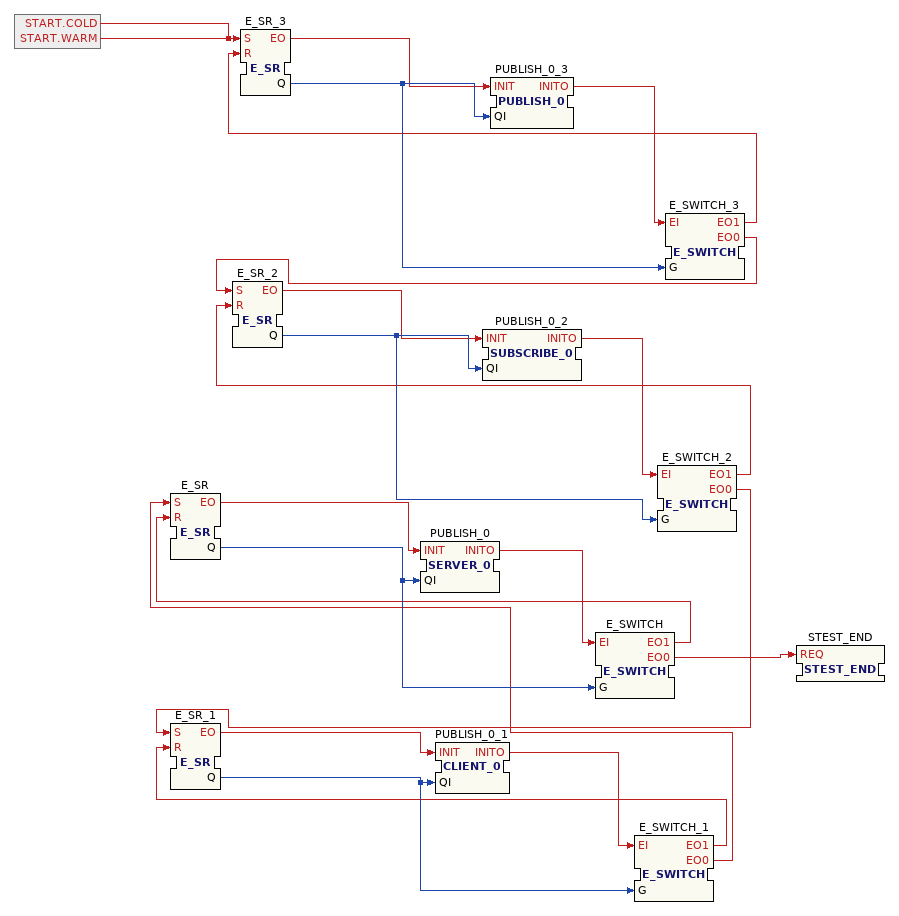
      FBS
        E_SR : E_SR;
        E_SWITCH : E_SWITCH;
        STEST_END : STEST_END;
        PUBLISH_0 : SERVER_0;
        E_SWITCH_1 : E_SWITCH;
        E_SR_1 : E_SR;
        E_SWITCH_2 : E_SWITCH;
        E_SR_2 : E_SR;
        E_SR_3 : E_SR;
        E_SWITCH_3 : E_SWITCH;
        PUBLISH_0_3 : PUBLISH_0;
        PUBLISH_0_2 : SUBSCRIBE_0;
        PUBLISH_0_1 : CLIENT_0;
      END_FBS
      EVENT_CONNECTIONS
        PUBLISH_0.INITO TO E_SWITCH.EI;
        E_SR_3.EO TO PUBLISH_0_3.INIT;
        PUBLISH_0_3.INITO TO E_SWITCH_3.EI;
        E_SR_2.EO TO PUBLISH_0_2.INIT;
        PUBLISH_0_2.INITO TO E_SWITCH_2.EI;
        E_SR_1.EO TO PUBLISH_0_1.INIT;
        PUBLISH_0_1.INITO TO E_SWITCH_1.EI;
        START.COLD TO E_SR_3.S;
        START.WARM TO E_SR_3.S;
        E_SWITCH_3.EO1 TO E_SR_3.R;
        E_SWITCH_3.EO0 TO E_SR_2.S;
        E_SWITCH_2.EO1 TO E_SR_2.R;
        E_SWITCH_2.EO0 TO E_SR_1.S;
        E_SWITCH_1.EO1 TO E_SR_1.R;
        E_SWITCH_1.EO0 TO E_SR.S;
        E_SWITCH.EO1 TO E_SR.R;
        E_SWITCH.EO0 TO STEST_END.REQ;
        E_SR.EO TO PUBLISH_0.INIT;
      END_CONNECTIONS
      DATA_CONNECTIONS
        E_SR.Q TO E_SWITCH.G;
        E_SR.Q TO PUBLISH_0.QI;
        E_SR_1.Q TO E_SWITCH_1.G;
        E_SR_2.Q TO E_SWITCH_2.G;
        E_SR_3.Q TO E_SWITCH_3.G;
        E_SR_3.Q TO PUBLISH_0_3.QI;
        E_SR_2.Q TO PUBLISH_0_2.QI;
        E_SR_1.Q TO PUBLISH_0_1.QI;
      END_CONNECTIONS
    END_RESOURCE
  END_DEVICE
  DEVICE Client : FORTE_PC(MGR_ID := "localhost:61499")
    {SET_ATTRIBUTE(Profile, HOLOBLOC)} (* device profile *)
    RESOURCE simpleClientTest : EMB_RES
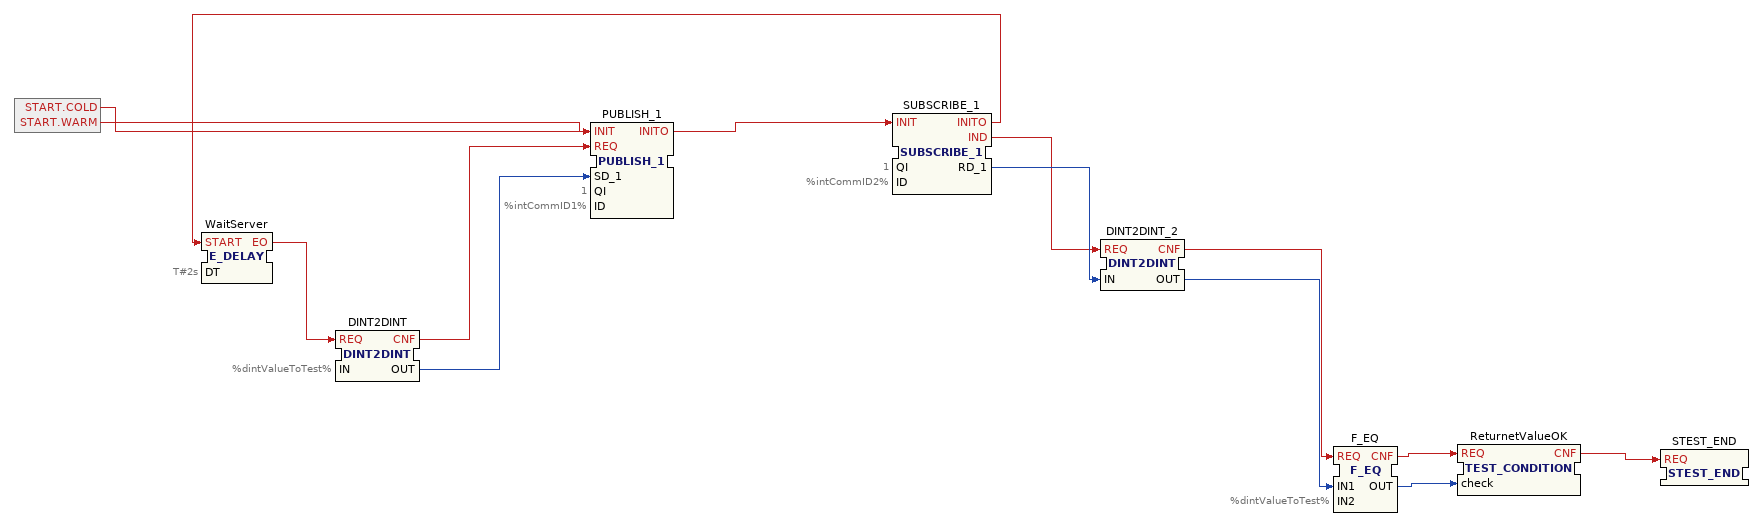
      FBS
        PUBLISH_1 : PUBLISH_1(QI := 1, ID := %intCommID1%);
        SUBSCRIBE_1 : SUBSCRIBE_1(QI := 1, ID := %intCommID2%);
        WaitServer : E_DELAY(DT := T#2s);
        ReturnetValueOK : TEST_CONDITION;
        F_EQ : F_EQ(IN2 := %dintValueToTest%);
        STEST_END : STEST_END;
        DINT2DINT : DINT2DINT(IN := %dintValueToTest%);
        DINT2DINT_2 : DINT2DINT;
      END_FBS
      EVENT_CONNECTIONS
        START.COLD TO PUBLISH_1.INIT;
        START.WARM TO PUBLISH_1.INIT;
        PUBLISH_1.INITO TO SUBSCRIBE_1.INIT;
        SUBSCRIBE_1.INITO TO WaitServer.START;
        DINT2DINT.CNF TO PUBLISH_1.REQ;
        F_EQ.CNF TO ReturnetValueOK.REQ;
        ReturnetValueOK.CNF TO STEST_END.REQ;
        WaitServer.EO TO DINT2DINT.REQ;
        DINT2DINT_2.CNF TO F_EQ.REQ;
        SUBSCRIBE_1.IND TO DINT2DINT_2.REQ;
      END_CONNECTIONS
      DATA_CONNECTIONS
        DINT2DINT.OUT TO PUBLISH_1.SD_1;
        F_EQ.OUT TO ReturnetValueOK.check;
        DINT2DINT_2.OUT TO F_EQ.IN1;
        SUBSCRIBE_1.RD_1 TO DINT2DINT_2.IN;
      END_CONNECTIONS
    END_RESOURCE
    RESOURCE multiDeviceStart : EMB_RES
